/// This function block is a container for equipment that is used by this unit.
/// Equipment is grouped by its kind (actuator, axes, io, ...).
/// It extends from [ManagedObjectContainer](xref:ZCore.ManagedObjectContainer) such that the parent
/// (= the unit itself) can be passed to equipment instances.
FUNCTION_BLOCK TransportEquipment EXTENDS TransportContainer
VAR_INPUT
  Io : TransportIo(_parent);
  Actuator : TransportActuator(_parent);
  Axis : TransportAxis(_parent);
  Fieldbus : TransportFieldbus(_parent);
  Unit : TransportLinkedUnit(_parent);
END_VAR

END_FUNCTION_BLOCK

(* stored: Version 1.1.0.1
   POU TransportEquipment: Id {8f0855ff-f26a-46ae-8f7e-b63dfcbe8283}, SpecialFunc None *)
